// TIA Portal project "elektro_boiler" (V16)

(* hardware
DEVICE "S7-1200 station_1"  S7-1200 Station
   slot 0: "Rack_0"  S7-1200 Rack  Rack  V1.0
   slot 1: "PLC_1"  CPU 1215C DC/DC/Rly  6ES7 215-1HG40-0XB0  V4.4
   slot 2: "DQ 8x24VDC _1"  SM 1222 DQ8 x 24VDC  6ES7 222-1BF30-0XB0  V1.0
   slot 3: "AI 8x13BIT_1"  6ES7 231-4HF32-0XB0  V2.1
*)

// ===== PLC "PLC_1"  CPU 1215C DC/DC/Rly =====

VAR_GLOBAL   // PLC tag table "Default tag table"
   "Clock_Byte" AT %MB0 : Byte;
   "Clock_10Hz" AT %M0.0 : Bool;
   "Clock_5Hz" AT %M0.1 : Bool;
   "Clock_2.5Hz" AT %M0.2 : Bool;
   "Clock_2Hz" AT %M0.3 : Bool;
   "Clock_1.25Hz" AT %M0.4 : Bool;
   "Clock_1Hz" AT %M0.5 : Bool;
   "Clock_0.625Hz" AT %M0.6 : Bool;
   "Clock_0.5Hz" AT %M0.7 : Bool;
   "TRUE" AT %M5.1 : Bool;
   "FALSE" AT %M5.0 : Bool;
   "puls_1_sec_t" AT %M4.0 : Bool;
   "puls_1_sec" AT %M4.1 : Bool;
   "EVEN" AT %M4.2 : Bool;
   "ODD" AT %M4.3 : Bool;
END_VAR

VAR_GLOBAL   // PLC tag table "DO"
   "ELECTR_DO_1" AT %Q0.0 : Bool;
   "ELECTR_DO_2" AT %Q0.1 : Bool;
   "ELECTR_DO_3" AT %Q0.2 : Bool;
   "ELECTR_DO_4" AT %Q0.3 : Bool;
   "ELECTR_DO_5" AT %Q0.4 : Bool;
   "ELECTR_DO_6" AT %Q0.5 : Bool;
   "ELECTR_DO_7" AT %Q0.6 : Bool;
   "ELECTR_DO_8" AT %Q0.7 : Bool;
   "PUMP1" AT %Q1.0 : Bool;
   "PUMP2" AT %Q1.1 : Bool;
END_VAR

VAR_GLOBAL   // PLC tag table "AI"
   "TEMP_IN" AT %IW112 : Int;
   "TEMP_OUT" AT %IW114 : Int;
   "PRESSURE" AT %IW116 : Int;
   "CURRENT_A" AT %IW118 : Int;
   "CURRENT_B" AT %IW120 : Int;
   "CURRENT_C" AT %IW122 : Int;
END_VAR

TYPE "AIN"
   STRUCT
      data_raw : Int;   // Сырое значение
      signal : Real;   // Значение сигнала в электрических единицах (мА, В и т.д.)
      eng : Real;   // Масштабированное значение аналогового сигнала
      status_0 : Bool;   // Неисправность канала
      status_1 : Bool;   // Ошибка калибровки (CalFault)
      status_2 : Bool;   // Выше HH
      status_3 : Bool;   // Выше H
      status_4 : Bool;   // Ниже L
      status_5 : Bool;   // Ниже LL
      status_6 : Bool;   // Резерв.
      status_7 : Bool;   // Выше диапазона (OverRange)
      status_8 : Bool;   // Ниже диапазона (UnderRange
      status_9 : Bool;   // Выше шкалы (OverScale)
      status_10 : Bool;   // Ниже шкалы (UnderScale)
      status_11 : Bool;   // Резерв.
      status_12 : Bool;   // Резерв.
      status_13 : Bool;   // Резерв.
      status_14 : Bool;   // Маскирование сигнала включено
      status_15 : Bool;   // Имитация сигнала включена
      SclMax : Real;   // Максимальное значение шкалы сигнала (в инженерных
      SclMin : Real;   // Минимальное значение шкалы сигнала (в инженерных
      DeadBand : Real;   // Значение уставки зоны нечувствительности (в инженерных
      LL : Real;   // Значение уставки LL (в инженерных единицах)
      L : Real;   // Значение уставки L (в инженерных единицах)
      H : Real := 90.0;   // Значение уставки H (в инженерных единицах)
      HH : Real := 100.0;   // Значение уставки HH (в инженерных единицах)
      config_0 : Bool;   // Команда: включить имитацию аналогового сигнала
      config_1 : Bool;   // Зарезервировано
      config_2 : Bool;   // Команда: включить в обработку уставку LL
      config_3 : Bool;   // Команда: включить в обработку уставку L
      config_4 : Bool;   // Команда: включить в обработку уставку H
      config_5 : Bool;   // Команда: включить в обработку уставку HH
      config_6 : Bool;   // Зарезервировано
      config_7 : Bool;   // Не используется
      config_8 : Bool;   // Команда: включить маскирование сигнала
      descID : Int;   // ID описания
   END_STRUCT;
END_TYPE

DATA_BLOCK "AINS_settings"   // DB1
{ S7_Optimized_Access := 'TRUE' }
VERSION : 0.1
   VAR
      UnderRange_limit : Real;
      UnderScale_limit : Real := 4.0;
      OverScale_limit : Real := 20.0;
      OverRange_limit : Real;
      analog_group : Int;
   END_VAR
BEGIN
END_DATA_BLOCK

DATA_BLOCK "AINS"   // DB2
{ S7_Optimized_Access := 'TRUE' }
VERSION : 0.1
   VAR RETAIN
      TEMP_IN_DB : "AIN";
      TEMP_OUT_DB : "AIN";
      PRESSURE_DB : "AIN";
      TEMPER_IN_3 : "AIN";
      TEMPER_IN_4 : "AIN";
      CHANGE_TIME : DWord;
   END_VAR
   VAR
      T_SETPOINT : Real;
      DEADBAND : Real;
   END_VAR
BEGIN
END_DATA_BLOCK

FUNCTION "AINS_general" : Void   // FC1, LAD
{ S7_Optimized_Access := 'TRUE' }
VERSION : 0.1
   VAR_INPUT
      UnderRange_limit : DInt;   // Ниже диапазона (UnderRange)
      UnderScale_limit : Real;   // Ниже шкалы (UnderScale)
      OverScale_limit : Real;   // Выше шкалы (OverScale)
      OverRange_limit : Real;   // Выше диапазона (OverRange)
      raw : Int;
   END_VAR
   VAR_IN_OUT
      AIN : "AIN";
   END_VAR
   VAR_TEMP
      UnderRange : Bool;
      OverRange : Bool;
      "a" : Real;
      "b" : Real;
      ChType1_0 : Bool;
      ChType1_1 : Bool;
      ChType1_2 : Bool;
      ChType1_3 : Bool;
      ChType1_4 : Bool;
      ChType1_5 : Bool;
      ChType1_6 : Bool;
      ChType1_7 : Bool;
      ChType1_8 : Bool;
      ChType1_9 : Bool;
      ChType1_10 : Bool;
      ChType1_11 : Bool;
      ChType1_12 : Bool;
      ChType1_13 : Bool;
      ChType1_14 : Bool;
      ChType1_15 : Bool;
      TEMPBOOL : Bool;
      doubletemp : DInt;
   END_VAR
   VAR_TEMP   // added for the SCL form of the ladder/FBD networks
      _w1 : Bool;
   END_VAR
BEGIN

REGION Network 1: Неисправность канала
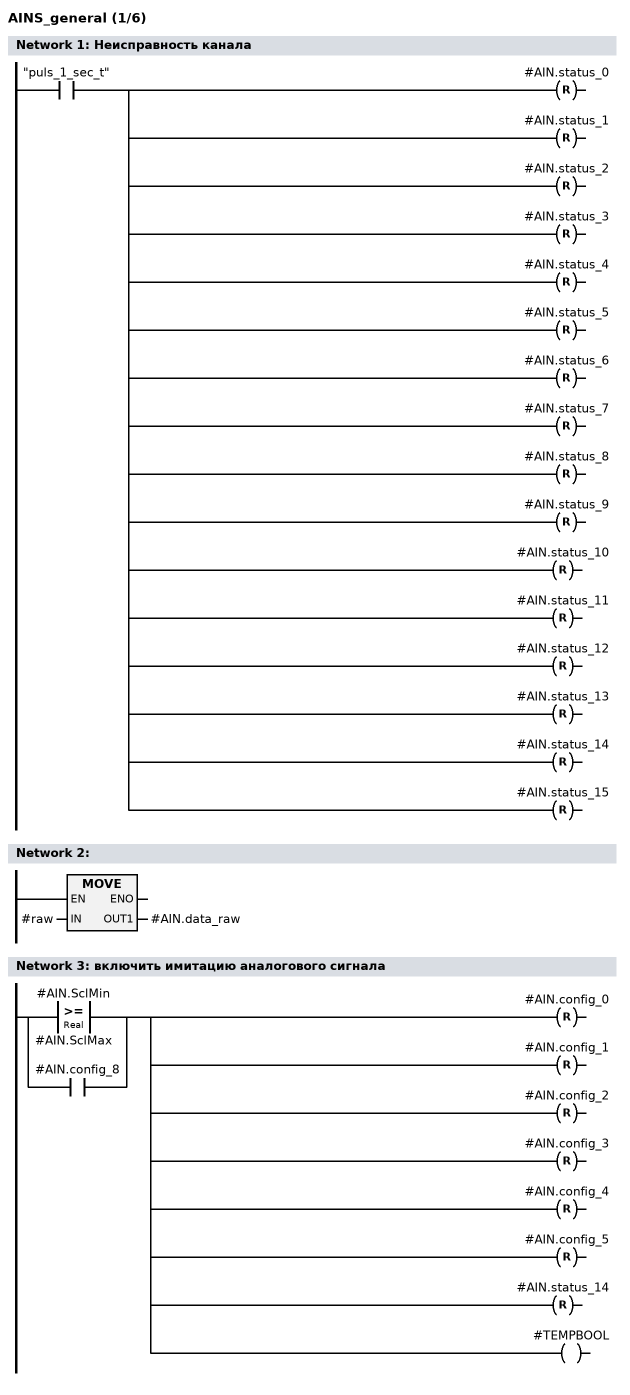
   RUNG wire#powerrail
      Contact( "puls_1_sec_t" )
      wire#w1
      R_Coil( #AIN.status_0 )
   END_RUNG
   RUNG wire#w1
      R_Coil( #AIN.status_1 )
   END_RUNG
   RUNG wire#w1
      R_Coil( #AIN.status_2 )
   END_RUNG
   RUNG wire#w1
      R_Coil( #AIN.status_3 )
   END_RUNG
   RUNG wire#w1
      R_Coil( #AIN.status_4 )
   END_RUNG
   RUNG wire#w1
      R_Coil( #AIN.status_5 )
   END_RUNG
   RUNG wire#w1
      R_Coil( #AIN.status_6 )
   END_RUNG
   RUNG wire#w1
      R_Coil( #AIN.status_7 )
   END_RUNG
   RUNG wire#w1
      R_Coil( #AIN.status_8 )
   END_RUNG
   RUNG wire#w1
      R_Coil( #AIN.status_9 )
   END_RUNG
   RUNG wire#w1
      R_Coil( #AIN.status_10 )
   END_RUNG
   RUNG wire#w1
      R_Coil( #AIN.status_11 )
   END_RUNG
   RUNG wire#w1
      R_Coil( #AIN.status_12 )
   END_RUNG
   RUNG wire#w1
      R_Coil( #AIN.status_13 )
   END_RUNG
   RUNG wire#w1
      R_Coil( #AIN.status_14 )
   END_RUNG
   RUNG wire#w1
      R_Coil( #AIN.status_15 )
   END_RUNG
   // the same network as SCL:
   IF "puls_1_sec_t" THEN
       #AIN.status_0 := FALSE;
       #AIN.status_1 := FALSE;
       #AIN.status_2 := FALSE;
       #AIN.status_3 := FALSE;
       #AIN.status_4 := FALSE;
       #AIN.status_5 := FALSE;
       #AIN.status_6 := FALSE;
       #AIN.status_7 := FALSE;
       #AIN.status_8 := FALSE;
       #AIN.status_9 := FALSE;
       #AIN.status_10 := FALSE;
       #AIN.status_11 := FALSE;
       #AIN.status_12 := FALSE;
       #AIN.status_13 := FALSE;
       #AIN.status_14 := FALSE;
       #AIN.status_15 := FALSE;
   END_IF;
END_REGION

REGION Network 2
   RUNG wire#powerrail
      Move(in := #raw, out1 => #AIN.data_raw)
   END_RUNG
   // the same network as SCL:
   #AIN.data_raw := #raw;
END_REGION

REGION Network 3: включить имитацию аналогового сигнала
   RUNG wire#powerrail
      { S7_Templates := "SrcType := Real" } GE_Contact(in1 := #AIN.SclMin, in2 := #AIN.SclMax)
      wire#w1
      R_Coil( #AIN.config_0 )
   END_RUNG
   RUNG wire#powerrail
      Contact( #AIN.config_8 )
   END_RUNG wire#w1
   RUNG wire#w1
      R_Coil( #AIN.config_1 )
   END_RUNG
   RUNG wire#w1
      R_Coil( #AIN.config_2 )
   END_RUNG
   RUNG wire#w1
      R_Coil( #AIN.config_3 )
   END_RUNG
   RUNG wire#w1
      R_Coil( #AIN.config_4 )
   END_RUNG
   RUNG wire#w1
      R_Coil( #AIN.config_5 )
   END_RUNG
   RUNG wire#w1
      R_Coil( #AIN.status_14 )
   END_RUNG
   RUNG wire#w1
      Coil( #TEMPBOOL )
   END_RUNG
   // the same network as SCL:
   #_w1 := (#AIN.SclMin >= #AIN.SclMax) OR #AIN.config_8;
   IF #_w1 THEN
       #AIN.config_0 := FALSE;
       #AIN.config_1 := FALSE;
       #AIN.config_2 := FALSE;
       #AIN.config_3 := FALSE;
       #AIN.config_4 := FALSE;
       #AIN.config_5 := FALSE;
       #AIN.status_14 := FALSE;
   END_IF;
   #TEMPBOOL := #_w1;
END_REGION

REGION Network 4
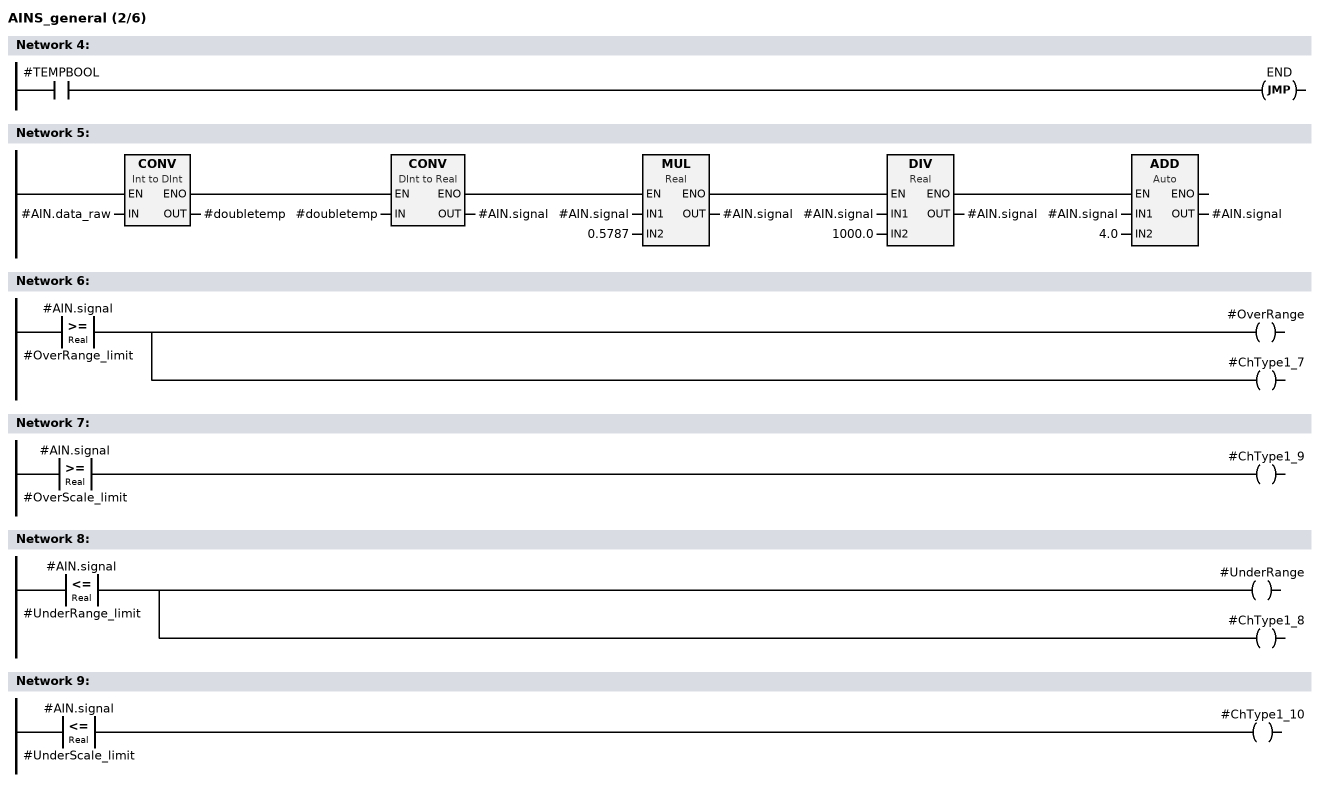
   RUNG wire#powerrail
      Contact( #TEMPBOOL )
      JumpCoil( END )
   END_RUNG
   // the same network as SCL:
   IF #TEMPBOOL THEN GOTO END; END_IF;
END_REGION

REGION Network 5
   RUNG wire#powerrail
      { S7_Templates := "[SrcType := Int, DestType := DInt]" } Convert(in := #AIN.data_raw, out => #doubletemp)
      { S7_Templates := "[SrcType := DInt, DestType := Real]" } Convert(in := #doubletemp, out => #AIN.signal)
      { S7_Templates := "SrcType := Real" } Mul(in1 := #AIN.signal, in2 := 0.5787, out => #AIN.signal)
      { S7_Templates := "SrcType := Real" } Div(in1 := #AIN.signal, in2 := 1000.0, out => #AIN.signal)
      Add(in1 := #AIN.signal, in2 := 4.0, out => #AIN.signal)
   END_RUNG
   // the same network as SCL:
   #doubletemp := INT_TO_DINT(#AIN.data_raw);
   #AIN.signal := DINT_TO_REAL(#doubletemp);
   #AIN.signal := #AIN.signal * 0.5787;
   #AIN.signal := #AIN.signal / 1000.0;
   #AIN.signal := #AIN.signal + 4.0;
END_REGION

REGION Network 6
   RUNG wire#powerrail
      { S7_Templates := "SrcType := Real" } GE_Contact(in1 := #AIN.signal, in2 := #OverRange_limit)
      wire#w1
      Coil( #OverRange )
   END_RUNG
   RUNG wire#w1
      Coil( #ChType1_7 )
   END_RUNG
   // the same network as SCL:
   #OverRange := #AIN.signal >= #OverRange_limit;
   #ChType1_7 := #OverRange;
END_REGION

REGION Network 7
   RUNG wire#powerrail
      { S7_Templates := "SrcType := Real" } GE_Contact(in1 := #AIN.signal, in2 := #OverScale_limit)
      Coil( #ChType1_9 )
   END_RUNG
   // the same network as SCL:
   #ChType1_9 := #AIN.signal >= #OverScale_limit;
END_REGION

REGION Network 8
   RUNG wire#powerrail
      { S7_Templates := "SrcType := Real" } LE_Contact(in1 := #AIN.signal, in2 := #UnderRange_limit)
      wire#w1
      Coil( #UnderRange )
   END_RUNG
   RUNG wire#w1
      Coil( #ChType1_8 )
   END_RUNG
   // the same network as SCL:
   #UnderRange := #AIN.signal <= #UnderRange_limit;
   #ChType1_8 := #UnderRange;
END_REGION

REGION Network 9
   RUNG wire#powerrail
      { S7_Templates := "SrcType := Real" } LE_Contact(in1 := #AIN.signal, in2 := #UnderScale_limit)
      Coil( #ChType1_10 )
   END_RUNG
   // the same network as SCL:
   #ChType1_10 := #AIN.signal <= #UnderScale_limit;
END_REGION

REGION Network 10
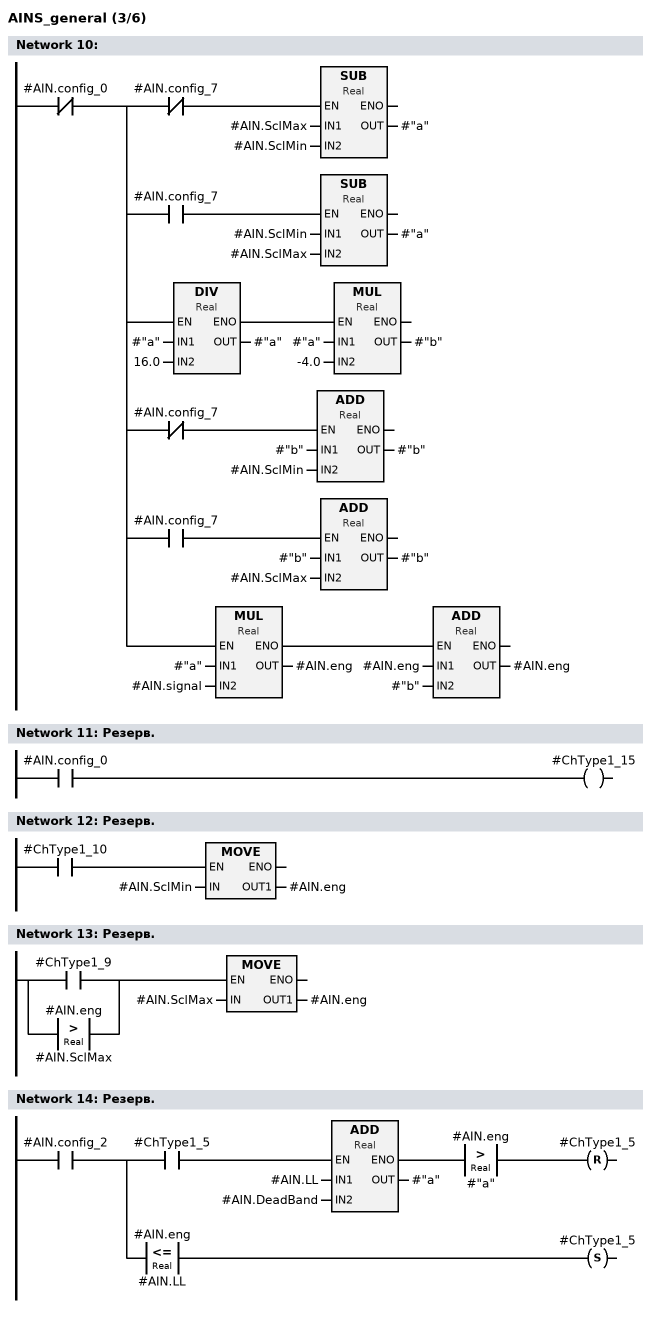
   RUNG wire#powerrail
      I_Contact( #AIN.config_0 )
      wire#w1
      I_Contact( #AIN.config_7 )
      { S7_Templates := "SrcType := Real" } Sub(in1 := #AIN.SclMax, in2 := #AIN.SclMin, out => #"a")
   END_RUNG
   RUNG wire#w1
      Contact( #AIN.config_7 )
      { S7_Templates := "SrcType := Real" } Sub(in1 := #AIN.SclMin, in2 := #AIN.SclMax, out => #"a")
   END_RUNG
   RUNG wire#w1
      { S7_Templates := "SrcType := Real" } Div(in1 := #"a", in2 := 16.0, out => #"a")
      { S7_Templates := "SrcType := Real" } Mul(in1 := #"a", in2 := -4.0, out => #"b")
   END_RUNG
   RUNG wire#w1
      I_Contact( #AIN.config_7 )
      { S7_Templates := "SrcType := Real" } Add(in1 := #"b", in2 := #AIN.SclMin, out => #"b")
   END_RUNG
   RUNG wire#w1
      Contact( #AIN.config_7 )
      { S7_Templates := "SrcType := Real" } Add(in1 := #"b", in2 := #AIN.SclMax, out => #"b")
   END_RUNG
   RUNG wire#w1
      { S7_Templates := "SrcType := Real" } Mul(in1 := #"a", in2 := #AIN.signal, out => #AIN.eng)
      { S7_Templates := "SrcType := Real" } Add(in1 := #AIN.eng, in2 := #"b", out => #AIN.eng)
   END_RUNG
   // the same network as SCL:
   IF NOT #AIN.config_0 AND NOT #AIN.config_7 THEN #"a" := #AIN.SclMax - #AIN.SclMin; END_IF;
   IF NOT #AIN.config_0 AND #AIN.config_7 THEN #"a" := #AIN.SclMin - #AIN.SclMax; END_IF;
   IF NOT #AIN.config_0 THEN
       #"a" := #"a" / 16.0;
       #"b" := #"a" * (-4.0);
   END_IF;
   IF NOT #AIN.config_0 AND NOT #AIN.config_7 THEN #"b" := #"b" + #AIN.SclMin; END_IF;
   IF NOT #AIN.config_0 AND #AIN.config_7 THEN #"b" := #"b" + #AIN.SclMax; END_IF;
   IF NOT #AIN.config_0 THEN
       #AIN.eng := #"a" * #AIN.signal;
       #AIN.eng := #AIN.eng + #"b";
   END_IF;
END_REGION

REGION Network 11: Резерв.
   RUNG wire#powerrail
      Contact( #AIN.config_0 )
      Coil( #ChType1_15 )
   END_RUNG
   // the same network as SCL:
   #ChType1_15 := #AIN.config_0;
END_REGION

REGION Network 12: Резерв.
   RUNG wire#powerrail
      Contact( #ChType1_10 )
      Move(in := #AIN.SclMin, out1 => #AIN.eng)
   END_RUNG
   // the same network as SCL:
   IF #ChType1_10 THEN #AIN.eng := #AIN.SclMin; END_IF;
END_REGION

REGION Network 13: Резерв.
   RUNG wire#powerrail
      Contact( #ChType1_9 )
      wire#w1
      Move(in := #AIN.SclMax, out1 => #AIN.eng)
   END_RUNG
   RUNG wire#powerrail
      { S7_Templates := "SrcType := Real" } GT_Contact(in1 := #AIN.eng, in2 := #AIN.SclMax)
   END_RUNG wire#w1
   // the same network as SCL:
   IF #ChType1_9 OR (#AIN.eng > #AIN.SclMax) THEN #AIN.eng := #AIN.SclMax; END_IF;
END_REGION

REGION Network 14: Резерв.
   RUNG wire#powerrail
      Contact( #AIN.config_2 )
      wire#w1
      Contact( #ChType1_5 )
      { S7_Templates := "SrcType := Real" } Add(in1 := #AIN.LL, in2 := #AIN.DeadBand, out => #"a")
      { S7_Templates := "SrcType := Real" } GT_Contact(in1 := #AIN.eng, in2 := #"a")
      R_Coil( #ChType1_5 )
   END_RUNG
   RUNG wire#w1
      { S7_Templates := "SrcType := Real" } LE_Contact(in1 := #AIN.eng, in2 := #AIN.LL)
      S_Coil( #ChType1_5 )
   END_RUNG
   // the same network as SCL:
   #_w1 := #AIN.config_2 AND #ChType1_5;
   IF #_w1 THEN #"a" := #AIN.LL + #AIN.DeadBand; END_IF;
   IF #_w1 AND (#AIN.eng > #"a") THEN #ChType1_5 := FALSE; END_IF;
   IF #AIN.config_2 AND (#AIN.eng <= #AIN.LL) THEN #ChType1_5 := TRUE; END_IF;
END_REGION

REGION Network 15: Резерв.
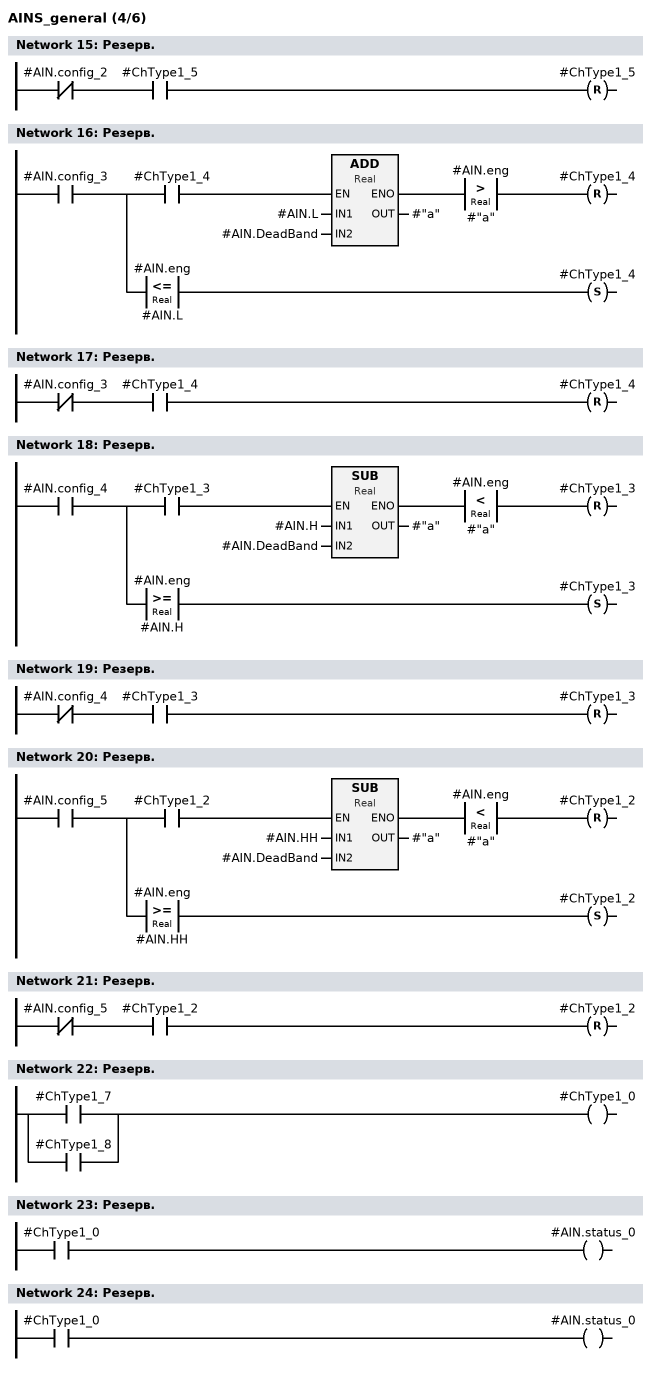
   RUNG wire#powerrail
      I_Contact( #AIN.config_2 )
      Contact( #ChType1_5 )
      R_Coil( #ChType1_5 )
   END_RUNG
   // the same network as SCL:
   IF NOT #AIN.config_2 AND #ChType1_5 THEN #ChType1_5 := FALSE; END_IF;
END_REGION

REGION Network 16: Резерв.
   RUNG wire#powerrail
      Contact( #AIN.config_3 )
      wire#w1
      Contact( #ChType1_4 )
      { S7_Templates := "SrcType := Real" } Add(in1 := #AIN.L, in2 := #AIN.DeadBand, out => #"a")
      { S7_Templates := "SrcType := Real" } GT_Contact(in1 := #AIN.eng, in2 := #"a")
      R_Coil( #ChType1_4 )
   END_RUNG
   RUNG wire#w1
      { S7_Templates := "SrcType := Real" } LE_Contact(in1 := #AIN.eng, in2 := #AIN.L)
      S_Coil( #ChType1_4 )
   END_RUNG
   // the same network as SCL:
   #_w1 := #AIN.config_3 AND #ChType1_4;
   IF #_w1 THEN #"a" := #AIN.L + #AIN.DeadBand; END_IF;
   IF #_w1 AND (#AIN.eng > #"a") THEN #ChType1_4 := FALSE; END_IF;
   IF #AIN.config_3 AND (#AIN.eng <= #AIN.L) THEN #ChType1_4 := TRUE; END_IF;
END_REGION

REGION Network 17: Резерв.
   RUNG wire#powerrail
      I_Contact( #AIN.config_3 )
      Contact( #ChType1_4 )
      R_Coil( #ChType1_4 )
   END_RUNG
   // the same network as SCL:
   IF NOT #AIN.config_3 AND #ChType1_4 THEN #ChType1_4 := FALSE; END_IF;
END_REGION

REGION Network 18: Резерв.
   RUNG wire#powerrail
      Contact( #AIN.config_4 )
      wire#w1
      Contact( #ChType1_3 )
      { S7_Templates := "SrcType := Real" } Sub(in1 := #AIN.H, in2 := #AIN.DeadBand, out => #"a")
      { S7_Templates := "SrcType := Real" } LT_Contact(in1 := #AIN.eng, in2 := #"a")
      R_Coil( #ChType1_3 )
   END_RUNG
   RUNG wire#w1
      { S7_Templates := "SrcType := Real" } GE_Contact(in1 := #AIN.eng, in2 := #AIN.H)
      S_Coil( #ChType1_3 )
   END_RUNG
   // the same network as SCL:
   #_w1 := #AIN.config_4 AND #ChType1_3;
   IF #_w1 THEN #"a" := #AIN.H - #AIN.DeadBand; END_IF;
   IF #_w1 AND (#AIN.eng < #"a") THEN #ChType1_3 := FALSE; END_IF;
   IF #AIN.config_4 AND (#AIN.eng >= #AIN.H) THEN #ChType1_3 := TRUE; END_IF;
END_REGION

REGION Network 19: Резерв.
   RUNG wire#powerrail
      I_Contact( #AIN.config_4 )
      Contact( #ChType1_3 )
      R_Coil( #ChType1_3 )
   END_RUNG
   // the same network as SCL:
   IF NOT #AIN.config_4 AND #ChType1_3 THEN #ChType1_3 := FALSE; END_IF;
END_REGION

REGION Network 20: Резерв.
   RUNG wire#powerrail
      Contact( #AIN.config_5 )
      wire#w1
      Contact( #ChType1_2 )
      { S7_Templates := "SrcType := Real" } Sub(in1 := #AIN.HH, in2 := #AIN.DeadBand, out => #"a")
      { S7_Templates := "SrcType := Real" } LT_Contact(in1 := #AIN.eng, in2 := #"a")
      R_Coil( #ChType1_2 )
   END_RUNG
   RUNG wire#w1
      { S7_Templates := "SrcType := Real" } GE_Contact(in1 := #AIN.eng, in2 := #AIN.HH)
      S_Coil( #ChType1_2 )
   END_RUNG
   // the same network as SCL:
   #_w1 := #AIN.config_5 AND #ChType1_2;
   IF #_w1 THEN #"a" := #AIN.HH - #AIN.DeadBand; END_IF;
   IF #_w1 AND (#AIN.eng < #"a") THEN #ChType1_2 := FALSE; END_IF;
   IF #AIN.config_5 AND (#AIN.eng >= #AIN.HH) THEN #ChType1_2 := TRUE; END_IF;
END_REGION

REGION Network 21: Резерв.
   RUNG wire#powerrail
      I_Contact( #AIN.config_5 )
      Contact( #ChType1_2 )
      R_Coil( #ChType1_2 )
   END_RUNG
   // the same network as SCL:
   IF NOT #AIN.config_5 AND #ChType1_2 THEN #ChType1_2 := FALSE; END_IF;
END_REGION

REGION Network 22: Резерв.
   RUNG wire#powerrail
      Contact( #ChType1_7 )
      wire#w1
      Coil( #ChType1_0 )
   END_RUNG
   RUNG wire#powerrail
      Contact( #ChType1_8 )
   END_RUNG wire#w1
   // the same network as SCL:
   #ChType1_0 := #ChType1_7 OR #ChType1_8;
END_REGION

REGION Network 23: Резерв.
   RUNG wire#powerrail
      Contact( #ChType1_0 )
      Coil( #AIN.status_0 )
   END_RUNG
   // the same network as SCL:
   #AIN.status_0 := #ChType1_0;
END_REGION

REGION Network 24: Резерв.
   RUNG wire#powerrail
      Contact( #ChType1_0 )
      Coil( #AIN.status_0 )
   END_RUNG
   // the same network as SCL:
   #AIN.status_0 := #ChType1_0;
END_REGION

REGION Network 25: Резерв.
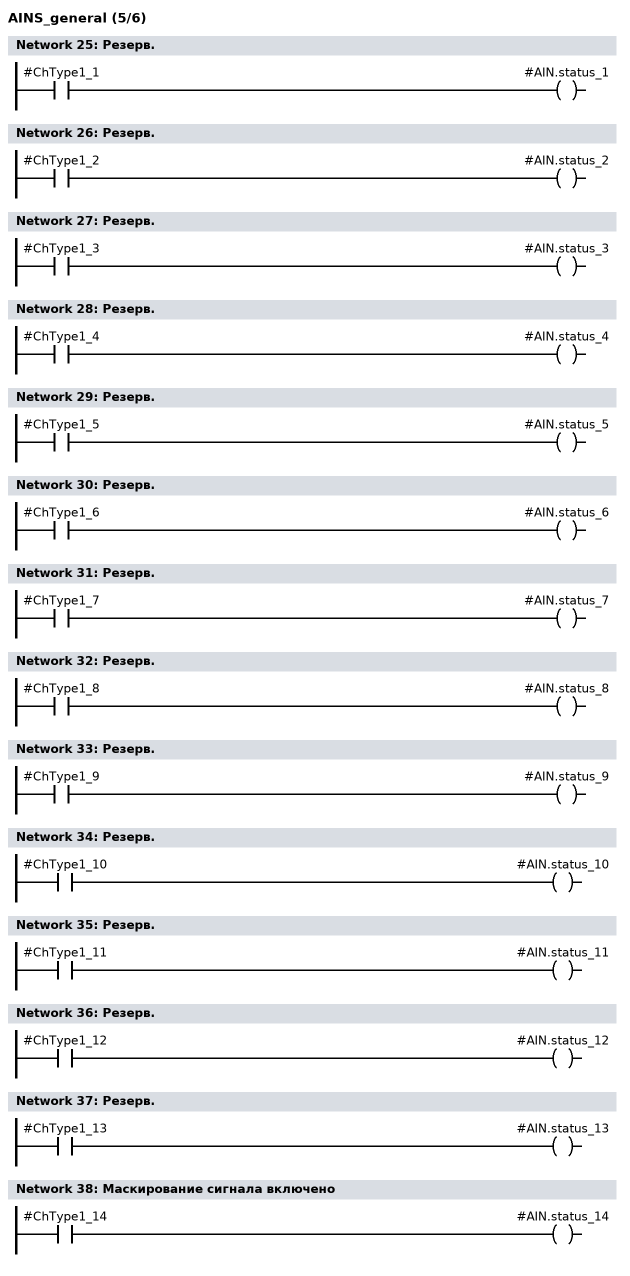
   RUNG wire#powerrail
      Contact( #ChType1_1 )
      Coil( #AIN.status_1 )
   END_RUNG
   // the same network as SCL:
   #AIN.status_1 := #ChType1_1;
END_REGION

REGION Network 26: Резерв.
   RUNG wire#powerrail
      Contact( #ChType1_2 )
      Coil( #AIN.status_2 )
   END_RUNG
   // the same network as SCL:
   #AIN.status_2 := #ChType1_2;
END_REGION

REGION Network 27: Резерв.
   RUNG wire#powerrail
      Contact( #ChType1_3 )
      Coil( #AIN.status_3 )
   END_RUNG
   // the same network as SCL:
   #AIN.status_3 := #ChType1_3;
END_REGION

REGION Network 28: Резерв.
   RUNG wire#powerrail
      Contact( #ChType1_4 )
      Coil( #AIN.status_4 )
   END_RUNG
   // the same network as SCL:
   #AIN.status_4 := #ChType1_4;
END_REGION

REGION Network 29: Резерв.
   RUNG wire#powerrail
      Contact( #ChType1_5 )
      Coil( #AIN.status_5 )
   END_RUNG
   // the same network as SCL:
   #AIN.status_5 := #ChType1_5;
END_REGION

REGION Network 30: Резерв.
   RUNG wire#powerrail
      Contact( #ChType1_6 )
      Coil( #AIN.status_6 )
   END_RUNG
   // the same network as SCL:
   #AIN.status_6 := #ChType1_6;
END_REGION

REGION Network 31: Резерв.
   RUNG wire#powerrail
      Contact( #ChType1_7 )
      Coil( #AIN.status_7 )
   END_RUNG
   // the same network as SCL:
   #AIN.status_7 := #ChType1_7;
END_REGION

REGION Network 32: Резерв.
   RUNG wire#powerrail
      Contact( #ChType1_8 )
      Coil( #AIN.status_8 )
   END_RUNG
   // the same network as SCL:
   #AIN.status_8 := #ChType1_8;
END_REGION

REGION Network 33: Резерв.
   RUNG wire#powerrail
      Contact( #ChType1_9 )
      Coil( #AIN.status_9 )
   END_RUNG
   // the same network as SCL:
   #AIN.status_9 := #ChType1_9;
END_REGION

REGION Network 34: Резерв.
   RUNG wire#powerrail
      Contact( #ChType1_10 )
      Coil( #AIN.status_10 )
   END_RUNG
   // the same network as SCL:
   #AIN.status_10 := #ChType1_10;
END_REGION

REGION Network 35: Резерв.
   RUNG wire#powerrail
      Contact( #ChType1_11 )
      Coil( #AIN.status_11 )
   END_RUNG
   // the same network as SCL:
   #AIN.status_11 := #ChType1_11;
END_REGION

REGION Network 36: Резерв.
   RUNG wire#powerrail
      Contact( #ChType1_12 )
      Coil( #AIN.status_12 )
   END_RUNG
   // the same network as SCL:
   #AIN.status_12 := #ChType1_12;
END_REGION

REGION Network 37: Резерв.
   RUNG wire#powerrail
      Contact( #ChType1_13 )
      Coil( #AIN.status_13 )
   END_RUNG
   // the same network as SCL:
   #AIN.status_13 := #ChType1_13;
END_REGION

REGION Network 38: Маскирование сигнала включено
   RUNG wire#powerrail
      Contact( #ChType1_14 )
      Coil( #AIN.status_14 )
   END_RUNG
   // the same network as SCL:
   #AIN.status_14 := #ChType1_14;
END_REGION

REGION Network 39: Имитация сигнала включена
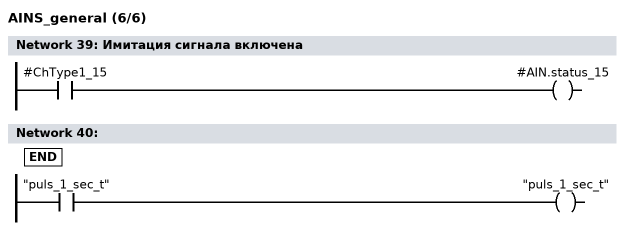
   RUNG wire#powerrail
      Contact( #ChType1_15 )
      Coil( #AIN.status_15 )
   END_RUNG
   // the same network as SCL:
   #AIN.status_15 := #ChType1_15;
END_REGION

REGION Network 40
   Label( END )
   RUNG wire#powerrail
      Contact( "puls_1_sec_t" )
      Coil( "puls_1_sec_t" )
   END_RUNG
   // the same network as SCL:
   END:
   "puls_1_sec_t" := "puls_1_sec_t";
END_REGION
END_FUNCTION

FUNCTION "AINS_main" : Void   // FC2, LAD
{ S7_Optimized_Access := 'TRUE' }
VERSION : 0.1
BEGIN

REGION Network 1
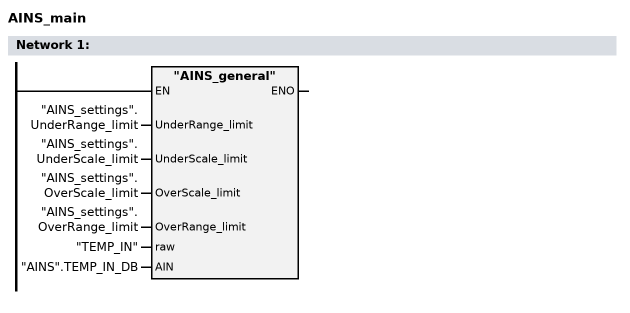
   RUNG wire#powerrail
      "AINS_general"(UnderRange_limit := "AINS_settings".UnderRange_limit, UnderScale_limit := "AINS_settings".UnderScale_limit, OverScale_limit := "AINS_settings".OverScale_limit, OverRange_limit := "AINS_settings".OverRange_limit, raw := "TEMP_IN", AIN := "AINS".TEMP_IN_DB)
   END_RUNG
   // the same network as SCL:
   "AINS_general"(UnderRange_limit := "AINS_settings".UnderRange_limit,
                  UnderScale_limit := "AINS_settings".UnderScale_limit,
                  OverScale_limit := "AINS_settings".OverScale_limit,
                  OverRange_limit := "AINS_settings".OverRange_limit,
                  raw := "TEMP_IN",
                  AIN := "AINS".TEMP_IN_DB);
END_REGION
END_FUNCTION

FUNCTION "Chang_general" : Void   // FC3, LAD
{ S7_Optimized_Access := 'TRUE' }
VERSION : 0.1
   VAR_INPUT
      SEKUNDS : DWord;
   END_VAR
   VAR_OUTPUT
      FIRST : Bool;
      SECOND : Bool;
   END_VAR
   VAR_TEMP
      SECOND_time : DWord;
      TMP : DWord;
   END_VAR
BEGIN

REGION Network 1
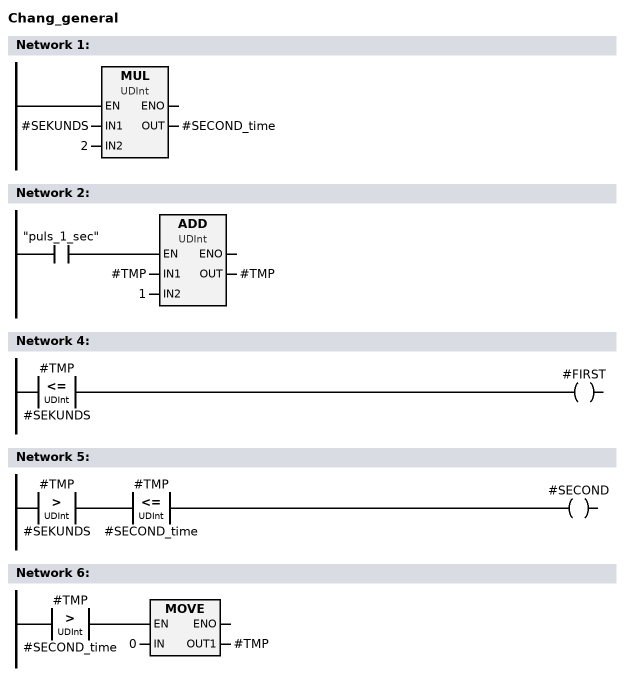
   RUNG wire#powerrail
      { S7_Templates := "SrcType := UDInt" } Mul(in1 := #SEKUNDS, in2 := 2, out => #SECOND_time)
   END_RUNG
   // the same network as SCL:
   #SECOND_time := #SEKUNDS * 2;
END_REGION

REGION Network 2
   RUNG wire#powerrail
      Contact( "puls_1_sec" )
      { S7_Templates := "SrcType := UDInt" } Add(in1 := #TMP, in2 := 1, out => #TMP)
   END_RUNG
   // the same network as SCL:
   IF "puls_1_sec" THEN #TMP := #TMP + 1; END_IF;
END_REGION

REGION Network 4
   RUNG wire#powerrail
      { S7_Templates := "SrcType := UDInt" } LE_Contact(in1 := #TMP, in2 := #SEKUNDS)
      Coil( #FIRST )
   END_RUNG
   // the same network as SCL:
   #FIRST := #TMP <= #SEKUNDS;
END_REGION

REGION Network 5
   RUNG wire#powerrail
      { S7_Templates := "SrcType := UDInt" } GT_Contact(in1 := #TMP, in2 := #SEKUNDS)
      { S7_Templates := "SrcType := UDInt" } LE_Contact(in1 := #TMP, in2 := #SECOND_time)
      Coil( #SECOND )
   END_RUNG
   // the same network as SCL:
   #SECOND := (#TMP > #SEKUNDS) AND (#TMP <= #SECOND_time);
END_REGION

REGION Network 6
   RUNG wire#powerrail
      { S7_Templates := "SrcType := UDInt" } GT_Contact(in1 := #TMP, in2 := #SECOND_time)
      Move(in := 0, out1 => #TMP)
   END_RUNG
   // the same network as SCL:
   IF #TMP > #SECOND_time THEN #TMP := 0; END_IF;
END_REGION
END_FUNCTION

FUNCTION "Cange_main" : Void   // FC4, LAD
{ S7_Optimized_Access := 'TRUE' }
VERSION : 0.1
BEGIN

REGION Network 1
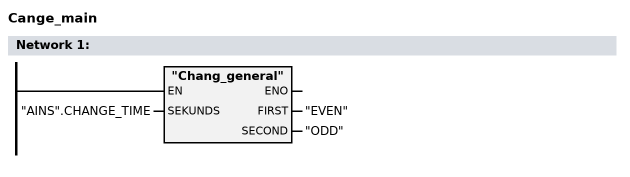
   RUNG wire#powerrail
      "Chang_general"(SEKUNDS := "AINS".CHANGE_TIME, FIRST => "EVEN", SECOND => "ODD")
   END_RUNG
   // the same network as SCL:
   "Chang_general"(SEKUNDS := "AINS".CHANGE_TIME, FIRST => "EVEN", SECOND => "ODD");
END_REGION
END_FUNCTION

FUNCTION "DOUT_general" : Void   // FC5, LAD
{ S7_Optimized_Access := 'TRUE' }
VERSION : 0.1
   VAR_INPUT
      AIN : Real;
      SET_POINT : Real;
      DEADBAND : Real;
   END_VAR
   VAR_OUTPUT
      OUT : Bool;
   END_VAR
   VAR_TEMP
      TEMPOR_MIN : Real;
      TEMPOR_MAX : Real;
   END_VAR
BEGIN

REGION Network 1
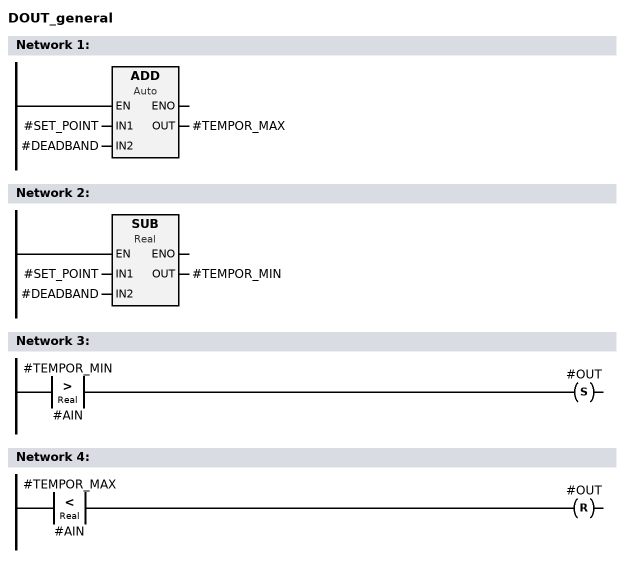
   RUNG wire#powerrail
      Add(in1 := #SET_POINT, in2 := #DEADBAND, out => #TEMPOR_MAX)
   END_RUNG
   // the same network as SCL:
   #TEMPOR_MAX := #SET_POINT + #DEADBAND;
END_REGION

REGION Network 2
   RUNG wire#powerrail
      { S7_Templates := "SrcType := Real" } Sub(in1 := #SET_POINT, in2 := #DEADBAND, out => #TEMPOR_MIN)
   END_RUNG
   // the same network as SCL:
   #TEMPOR_MIN := #SET_POINT - #DEADBAND;
END_REGION

REGION Network 3
   RUNG wire#powerrail
      { S7_Templates := "SrcType := Real" } GT_Contact(in1 := #TEMPOR_MIN, in2 := #AIN)
      S_Coil( #OUT )
   END_RUNG
   // the same network as SCL:
   IF #TEMPOR_MIN > #AIN THEN #OUT := TRUE; END_IF;
END_REGION

REGION Network 4
   RUNG wire#powerrail
      { S7_Templates := "SrcType := Real" } LT_Contact(in1 := #TEMPOR_MAX, in2 := #AIN)
      R_Coil( #OUT )
   END_RUNG
   // the same network as SCL:
   IF #TEMPOR_MAX < #AIN THEN #OUT := FALSE; END_IF;
END_REGION
END_FUNCTION

FUNCTION "DOUT_main" : Void   // FC6, LAD
{ S7_Optimized_Access := 'TRUE' }
VERSION : 0.1
   VAR_TEMP
      OUT : Bool;
   END_VAR
BEGIN

REGION Network 1
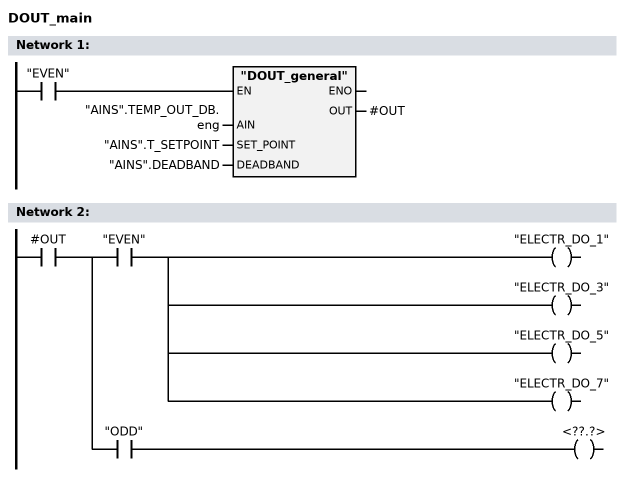
   RUNG wire#powerrail
      Contact( "EVEN" )
      "DOUT_general"(AIN := "AINS".TEMP_OUT_DB.eng, SET_POINT := "AINS".T_SETPOINT, DEADBAND := "AINS".DEADBAND, OUT => #OUT)
   END_RUNG
   // the same network as SCL:
   IF "EVEN" THEN
       "DOUT_general"(AIN := "AINS".TEMP_OUT_DB.eng,
                      SET_POINT := "AINS".T_SETPOINT,
                      DEADBAND := "AINS".DEADBAND,
                      OUT => #OUT);
   END_IF;
END_REGION

REGION Network 2
   RUNG wire#powerrail
      Contact( #OUT )
      wire#w1
      Contact( "EVEN" )
      wire#w2
      Coil( "ELECTR_DO_1" )
   END_RUNG
   RUNG wire#w2
      Coil( "ELECTR_DO_3" )
   END_RUNG
   RUNG wire#w2
      Coil( "ELECTR_DO_5" )
   END_RUNG
   RUNG wire#w2
      Coil( "ELECTR_DO_7" )
   END_RUNG
   RUNG wire#w1
      Contact( "ODD" )
      Coil(  )
   END_RUNG
   // the same network as SCL:
   "ELECTR_DO_1" := #OUT AND "EVEN";
   "ELECTR_DO_3" := "ELECTR_DO_1";
   "ELECTR_DO_5" := "ELECTR_DO_1";
   "ELECTR_DO_7" := "ELECTR_DO_1";
   <??.?> := #OUT AND "ODD";
END_REGION
END_FUNCTION

ORGANIZATION_BLOCK "Main"   // OB1, LAD, ProgramCycle
TITLE = "Main Program Sweep (Cycle)"
{ S7_Optimized_Access := 'TRUE' }
VERSION : 0.1
   VAR_INPUT
      Initial_Call : Bool;   // Initial call of this OB
      Remanence : Bool;   // =True, if remanent data are available
   END_VAR
   VAR_TEMP   // added for the SCL form of the ladder/FBD networks
      _w1 : Bool;
   END_VAR
BEGIN

REGION Network 1
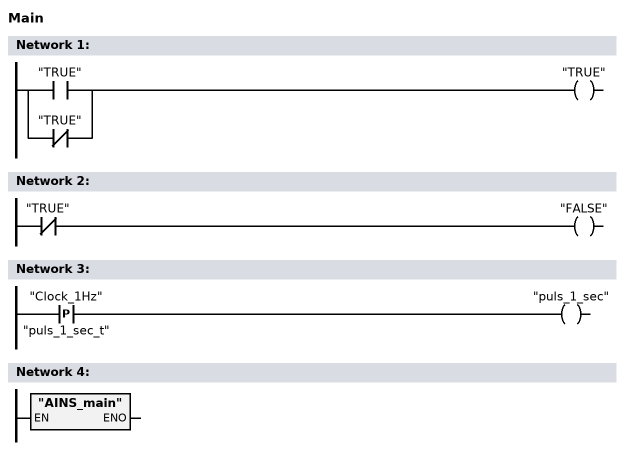
   RUNG wire#powerrail
      Contact( "TRUE" )
      wire#w1
      Coil( "TRUE" )
   END_RUNG
   RUNG wire#powerrail
      I_Contact( "TRUE" )
   END_RUNG wire#w1
   // the same network as SCL:
   "TRUE" := "TRUE" OR NOT "TRUE";
END_REGION

REGION Network 2
   RUNG wire#powerrail
      I_Contact( "TRUE" )
      Coil( "FALSE" )
   END_RUNG
   // the same network as SCL:
   "FALSE" := NOT "TRUE";
END_REGION

REGION Network 3
   RUNG wire#powerrail
      P_Contact(operand := "Clock_1Hz", bit := "puls_1_sec_t")
      Coil( "puls_1_sec" )
   END_RUNG
   // the same network as SCL:
   #_w1 := "Clock_1Hz" AND NOT "puls_1_sec_t";   // rising edge of "Clock_1Hz"
   "puls_1_sec_t" := "Clock_1Hz";
   "puls_1_sec" := #_w1;
END_REGION

REGION Network 4
   RUNG wire#powerrail
      "AINS_main"()
   END_RUNG
   // the same network as SCL:
   "AINS_main"();
END_REGION
END_ORGANIZATION_BLOCK